// Discards the current limit, returning the previous limit.
FUNCTION INTERNAL F_SbhPopLimit : HRESULT
VAR_IN_OUT
    stState     : ST_ParserInternalState;
END_VAR
VAR_INPUT
    nOldLimit   : UDINT;
END_VAR


stState.nCurrentLimit := nOldLimit;
F_SbhPopLimit := F_SbhRecomputeBufferSizeAfterLimit(stState);

END_FUNCTION

(* stored: Version 1.1.0.1
   POU F_SbhPopLimit: Id {754c0900-5e24-47a2-933a-820e2db1ac8f}, SpecialFunc None *)
